// TIA Portal V16 export
// export: Created 2024-09-05T17:36:34.2542997Z, ExportSetting WithDefaults, DisplayName Totally Integrated Automation Portal, DisplayVersion V16 Update 6, DisplayName TIA Portal Version Control Interface, DisplayVersion V16 Update 2, DisplayName TIA Portal Openness, DisplayVersion V16 Update 6, DisplayName STEP 7 Professional, DisplayVersion V16 Update 6, DisplayName STEP 7 Safety, DisplayVersion V16, DisplayName WinCC Advanced, DisplayVersion V16 Update 6
VAR_GLOBAL   // PLC tag table "Data Costant"
END_VAR
VAR_GLOBAL CONSTANT   // user constants
   MaxCreateNFP : Int := 5;
   MaxDataReading : Int := 25;
   MaxRoundNumber : Int := 1;
   NumberOfmessages : Int := 6;
   MaxStageStep : Int := 25;
   MaxInitStep : Int := 2;
   MaxRobot : Int := 3;
   "MaxReader(1)" : Int := 5;
   MaxSolenoid : Int := 48;
   NotUsed : Int := 0;
   MasterNFP : Int := 2;
   SecondaryNFP : Int := 3;
   Component : Int := 4;
END_VAR
